# EPICS autosave request: ioc/iocBoot/iocPico8/auto_settings.req
file "pico8_settings.req",          P=$(P),  R=det1:
file "NDStdArrays_settings.req",    P=$(P),  R=image1:
file "commonPlugin_settings.req",   P=$(P)
